Staubli VAL3: onEditItem.pgx

public program onEditItem(string& x_sEvent[] (dimensions=1), num x_nIndex (dimensions=1), num x_nIndexItem (dimensions=1))
begin
  // edit the custom element that was add in the list
  call onEditTrsf(x_nIndex,x_nIndexItem,x_sEvent)
end
